FUNCTION_BLOCK Linie
VAR_INPUT
	bEnable:BOOL;
	bStart:BOOL;
	bSensor_Vorne :BOOL;
	bSensor_Mitte :BOOL;
	bSensor_Hinten :BOOL;
END_VAR
VAR_OUTPUT
	bRollenStopper_Vorne :BOOL;
	bRollenStopper_Mitte :BOOL;	
	estate : E_State_Linie;
	estate_A1 :E_STATE_AMPEL;
	estate_A2 :E_STATE_AMPEL;
END_VAR
VAR
	T_enable:BOOL;
    tTimer : TON; // Timer Variable
END_VAR


tTimer(IN:=T_enable, PT:=T#1S);

IF NOT bEnable THEN
    eState := E_State_Linie.IDLE;
END_IF

CASE eState OF
    E_State_Linie.IDLE:
	
        IF bEnable THEN
            eState := E_State_Linie.INIT;
        END_IF

    E_State_Linie.INIT:

		//Ampel 1 Umschalten
		IF NOT bSensor_Vorne THEN
			estate_A1 :=E_STATE_AMPEL.YELLOW;
		ELSE
			estate_A1 :=E_STATE_AMPEL.GREEN;
		END_IF
		//Ampel 2 Umschalten
		IF  bSensor_Hinten THEN
			estate_A2 :=E_STATE_AMPEL.YELLOW;
		ELSE
			estate_A2 :=E_STATE_AMPEL.GREEN;
		END_IF
		
		IF NOT bSensor_Mitte AND bSensor_Vorne THEN
			eState := E_State_Linie.OPEN_START;
		ELSIF NOT bSensor_Mitte AND NOT bSensor_Vorne THEN
		 	eState:=E_State_Linie.WAIT_START;
		END_IF
		
	    IF bStart THEN
			eState:=E_State_Linie.START;
		END_IF
		
	E_State_Linie.START:
		//Ampel 1 Umschalten
		IF NOT bSensor_Vorne THEN
			estate_A1 :=E_STATE_AMPEL.YELLOW;
		ELSE
			estate_A1 :=E_STATE_AMPEL.GREEN;
		END_IF
		//Ampel 2 Umschalten
		
		IF  bSensor_Hinten THEN
			estate_A2 :=E_STATE_AMPEL.YELLOW;
		ELSE
			estate_A2 :=E_STATE_AMPEL.GREEN;
		END_IF
	
		IF bSensor_Hinten AND bSensor_Mitte THEN
			eState := E_State_Linie.WAIT_MIDLE;		
		ELSIF NOT bSensor_Hinten AND bSensor_Mitte THEN
			eState := E_State_Linie.OPEN_MIDLE;
		END_IF
		
	E_State_Linie.WAIT_MIDLE:
	
		estate_A2 :=E_STATE_AMPEL.RED;
		IF NOT bSensor_Hinten THEN
			eState := E_State_Linie.OPEN_MIDLE;
		END_IF

    E_State_Linie.OPEN_MIDLE:
	
		bRollenStopper_Mitte:=TRUE;
		IF NOT bSensor_Mitte THEN
			T_enable:=TRUE;
		END_IF
        IF tTimer.Q THEN
            eState := E_State_Linie.CLOSE_MIDLE;
			T_enable:=FALSE;
        END_IF

    E_State_Linie.CLOSE_MIDLE:
	
		bRollenStopper_Mitte:=FALSE;
        IF NOT bSensor_Mitte AND bSensor_Vorne THEN
            eState := E_State_Linie.OPEN_START;
		ELSIF NOT bSensor_Mitte AND NOT bSensor_Vorne THEN
			eState := E_State_Linie.WAIT_START;
        END_IF
		
	E_State_Linie.WAIT_START:
	
		estate_A1 :=E_STATE_AMPEL.RED;
        IF bSensor_Vorne THEN
            eState := E_State_Linie.OPEN_START;
        END_IF
		
    E_State_Linie.OPEN_START:
		bRollenStopper_Vorne:=TRUE;
		IF NOT bSensor_Vorne THEN
			T_enable:=TRUE;
		END_IF
        IF tTimer.Q THEN
            eState := E_State_Linie.CLOSE_START;
			T_enable:=FALSE;
        END_IF
		
    E_State_Linie.CLOSE_START:
	
		bRollenStopper_Vorne:=FALSE;
		IF bSensor_Mitte THEN
        	eState := E_State_Linie.DONE;
		END_IF	

    E_State_Linie.DONE:
    eState := E_State_Linie.IDLE;
	
END_CASE

END_FUNCTION_BLOCK

(* stored: Version 1.1.0.1, ProductVersion 3.1.4024.13
   POU Linie: Id {8cb3be87-1920-4ad8-9827-896f28ae3174}, SpecialFunc None *)
